(* PLC project Desconhecido, UFSCar Conversor PNML2Ladder 1 *)
(* stored: creationDateTime 2025-01-15T12:13:14, modificationDateTime 2025-02-12T16:48:13 *)

PROGRAM instance0

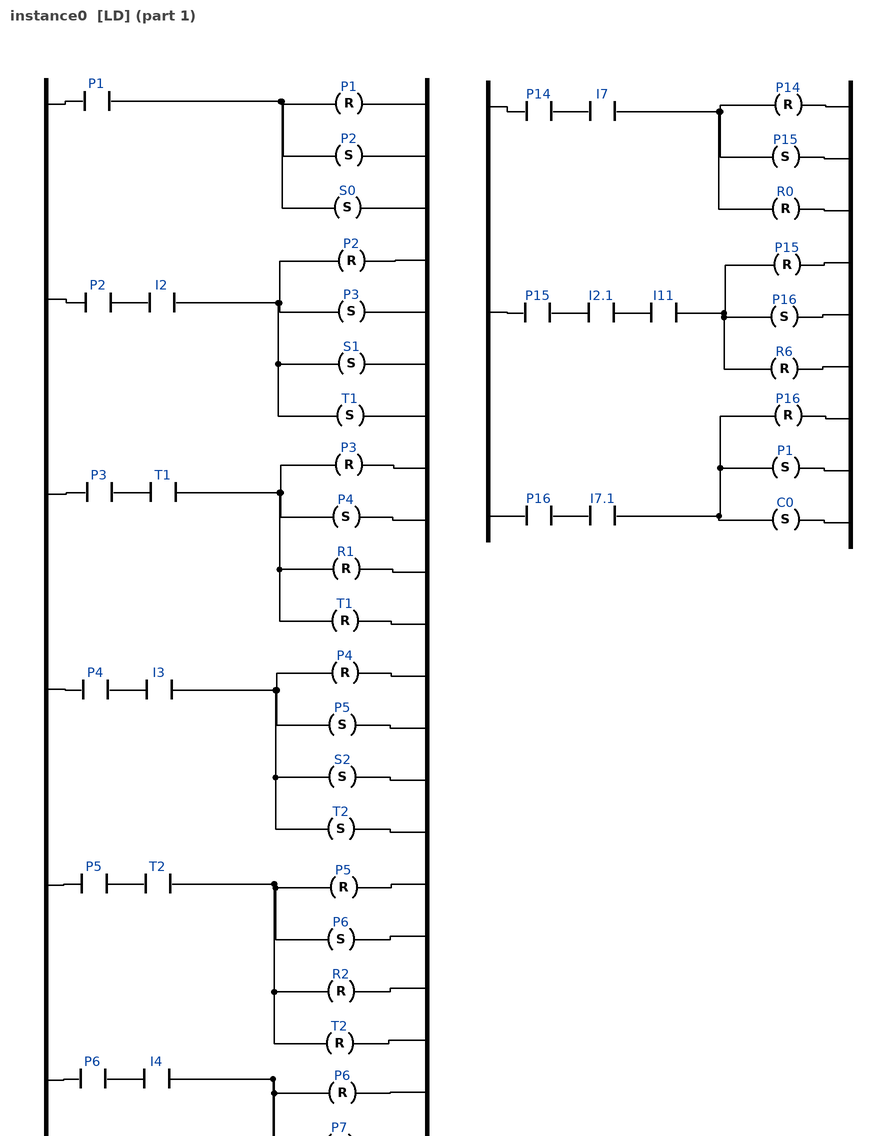
(* LD diagram, written out as Structured Text *)
IF P2 AND I2 THEN P2 := FALSE; END_IF;
IF P2 AND I2 THEN P3 := TRUE; END_IF;
IF P2 AND I2 THEN S1 := TRUE; END_IF;
IF P2 AND I2 THEN T1 := TRUE; END_IF;
IF P3 AND T1 THEN P4 := TRUE; END_IF;
IF P3 AND T1 THEN R1 := FALSE; END_IF;
IF P3 AND T1 THEN P3 := FALSE; END_IF;
IF P3 AND T1 THEN T1 := FALSE; END_IF;
IF P4 AND I3 THEN P4 := FALSE; END_IF;
IF P4 AND I3 THEN T2 := TRUE; END_IF;
IF P4 AND I3 THEN P5 := TRUE; END_IF;
IF P4 AND I3 THEN S2 := TRUE; END_IF;
IF P5 AND T2 THEN P5 := FALSE; END_IF;
IF P5 AND T2 THEN T2 := FALSE; END_IF;
IF P5 AND T2 THEN P6 := TRUE; END_IF;
IF P5 AND T2 THEN R2 := FALSE; END_IF;
IF P6 AND I4 THEN P6 := FALSE; END_IF;
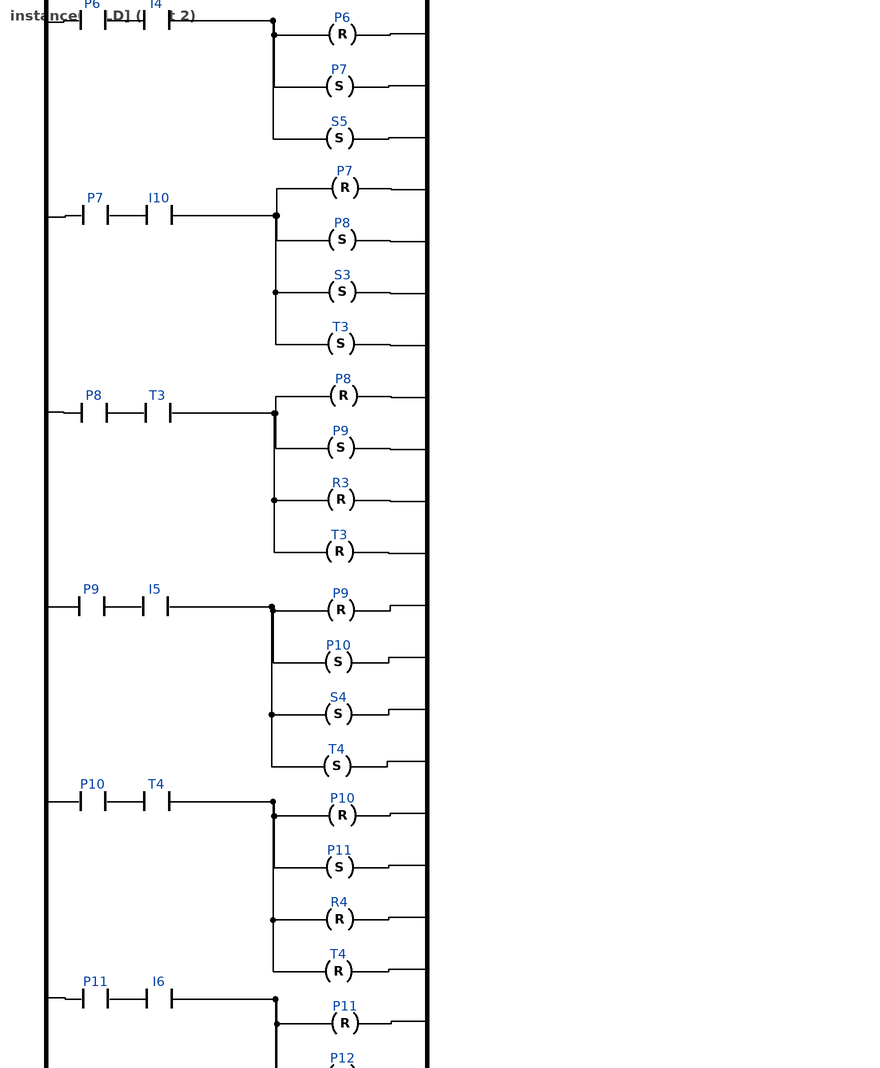
IF P6 AND I4 THEN P7 := TRUE; END_IF;
IF P6 AND I4 THEN S5 := TRUE; END_IF;
IF P1 THEN S0 := TRUE; END_IF;
IF P1 THEN P1 := FALSE; END_IF;
IF P1 THEN P2 := TRUE; END_IF;
IF P7 AND I10 THEN P7 := FALSE; END_IF;
IF P7 AND I10 THEN T3 := TRUE; END_IF;
IF P7 AND I10 THEN P8 := TRUE; END_IF;
IF P7 AND I10 THEN S3 := TRUE; END_IF;
IF P9 AND I5 THEN P9 := FALSE; END_IF;
IF P9 AND I5 THEN T4 := TRUE; END_IF;
IF P9 AND I5 THEN P10 := TRUE; END_IF;
IF P9 AND I5 THEN S4 := TRUE; END_IF;
IF P8 AND T3 THEN P8 := FALSE; END_IF;
IF P8 AND T3 THEN T3 := FALSE; END_IF;
IF P8 AND T3 THEN P9 := TRUE; END_IF;
IF P8 AND T3 THEN R3 := FALSE; END_IF;
IF P10 AND T4 THEN P10 := FALSE; END_IF;
IF P10 AND T4 THEN T4 := FALSE; END_IF;
IF P10 AND T4 THEN P11 := TRUE; END_IF;
IF P10 AND T4 THEN R4 := FALSE; END_IF;
IF P11 AND I6 THEN P11 := FALSE; END_IF;
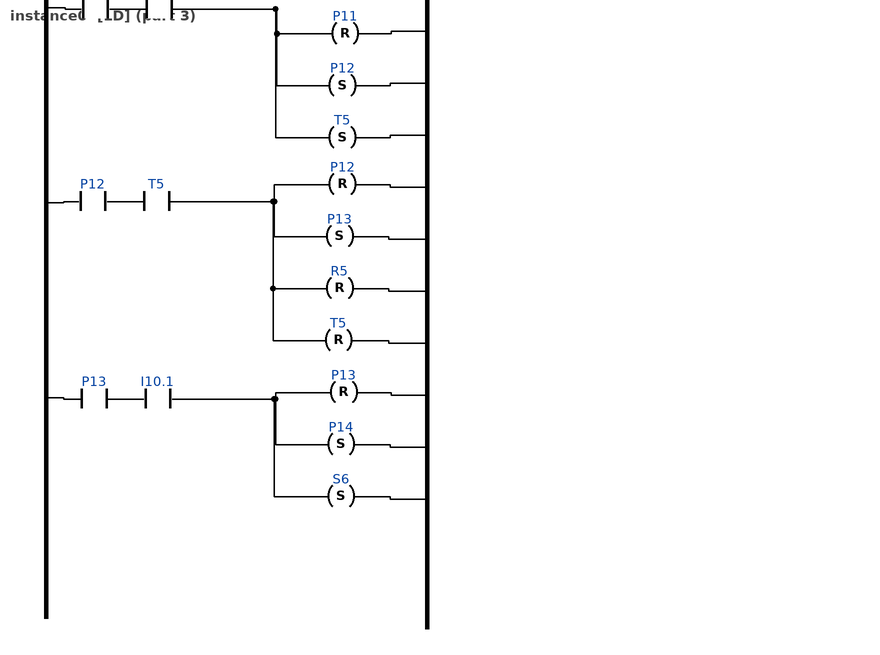
IF P11 AND I6 THEN P12 := TRUE; END_IF;
IF P11 AND I6 THEN T5 := TRUE; END_IF;
IF P13 AND I10.1 THEN P13 := FALSE; END_IF;
IF P13 AND I10.1 THEN P14 := TRUE; END_IF;
IF P13 AND I10.1 THEN S6 := TRUE; END_IF;
IF P12 AND T5 THEN P12 := FALSE; END_IF;
IF P12 AND T5 THEN T5 := FALSE; END_IF;
IF P12 AND T5 THEN P13 := TRUE; END_IF;
IF P12 AND T5 THEN R5 := FALSE; END_IF;
IF P14 AND I7 THEN P14 := FALSE; END_IF;
IF P14 AND I7 THEN P15 := TRUE; END_IF;
IF P14 AND I7 THEN R0 := FALSE; END_IF;
IF P15 AND I2.1 AND I11 THEN P15 := FALSE; END_IF;
IF P15 AND I2.1 AND I11 THEN P16 := TRUE; END_IF;
IF P15 AND I2.1 AND I11 THEN R6 := FALSE; END_IF;
IF P16 AND I7.1 THEN P16 := FALSE; END_IF;
IF P16 AND I7.1 THEN P1 := TRUE; END_IF;
IF P16 AND I7.1 THEN C0 := TRUE; END_IF;
END_PROGRAM

CONFIGURATION config0
  RESOURCE resource1 ON PLC
    TASK task0(INTERVAL := T#20ms, PRIORITY := 0);
    PROGRAM instance0 WITH task0 : program0;
  END_RESOURCE
END_CONFIGURATION
